FUNCTION_BLOCK StallDetection (* Template for a simple Basic Function Block Type *)
  (* Standard: 61499-2 *)
  (* Version 1.0, 2019-06-06, Robert *)
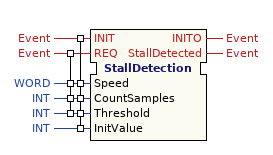
  EVENT_INPUT
    INIT WITH Speed, CountSamples, Threshold, InitValue; (* Initialization Request *)
    REQ WITH Speed, CountSamples, Threshold; (* Normal Execution Request *)
  END_EVENT
  EVENT_OUTPUT
    INITO; (* Initialization Confirm *)
    StallDetected;
  END_EVENT
  VAR_INPUT
    Speed : WORD; (* Input event qualifier *)
    CountSamples : INT;
    Threshold : INT;
    InitValue : INT;
  END_VAR
  VAR
    SampleArray : ARRAY [0..19] OF INT; (* Internal Variable *)
    currentSample : USINT; (* Internal Variable *)
    stalled : BOOL; (* Internal Variable *)
    sum : INT; (* Internal Variable *)
    i : USINT; (* Internal Variable *)
  END_VAR
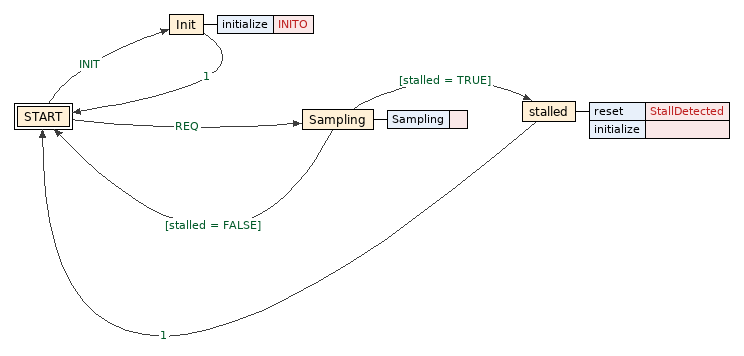
  EC_STATES
    START; (* Initial State *)
    Init : initialize -> INITO; (* Initialization *)
    stalled : reset -> StallDetected, initialize; (* Normal execution *)
    Sampling : Sampling;
  END_STATES
  EC_TRANSITIONS
    START TO Init := INIT;
    Sampling TO stalled := [stalled = TRUE];
    START TO Sampling := REQ;
    Sampling TO START := [stalled = FALSE];
    stalled TO START := 1;
    Init TO START := 1;
  END_TRANSITIONS
  ALGORITHM initialize IN ST: (* Initialization algorithm *)
FOR i:=0 TO 19 DO
	SampleArray[i]:= InitValue;
END_FOR;
  END_ALGORITHM
  ALGORITHM Sampling IN ST: (* Normally executed algorithm *)
IF currentSample < CountSamples  THEN
 currentSample := currentSample +1;
ELSE
 currentSample := 0;
END_IF;

SampleArray[currentSample] := Speed;

FOR i:=0 TO CountSamples DO
	sum := sum + SampleArray[i];
END_FOR;

sum := sum /CountSamples;

IF sum < Threshold THEN
	stalled := true;
	ELSE
	stalled := false;
END_IF;
  END_ALGORITHM
  ALGORITHM reset IN ST: (* new algorithm *)
stalled := false;
  END_ALGORITHM
END_FUNCTION_BLOCK
